PROGRAM OP90_MP_IO
VAR
	OP90_MP_DI_MODULE_1 AT %I* : WORD;
	OP90_MP_DI_MODULE_2 AT %I* : WORD;
	OP90_MP_DI_MODULE_3 AT %I* : WORD;
	
	OP90_MP_DO_MODULE_1 AT %Q* : WORD;
	OP90_MP_DO_MODULE_2 AT %Q* : WORD;
	
	WORD_AS_BIT_0: WORD_AS_BIT;
	WORD_AS_BIT_1: WORD_AS_BIT;
	WORD_AS_BIT_2: WORD_AS_BIT;
	
	BIT_AS_WORD_0: BIT_AS_WORD;
	BIT_AS_WORD_1: BIT_AS_WORD;
END_VAR

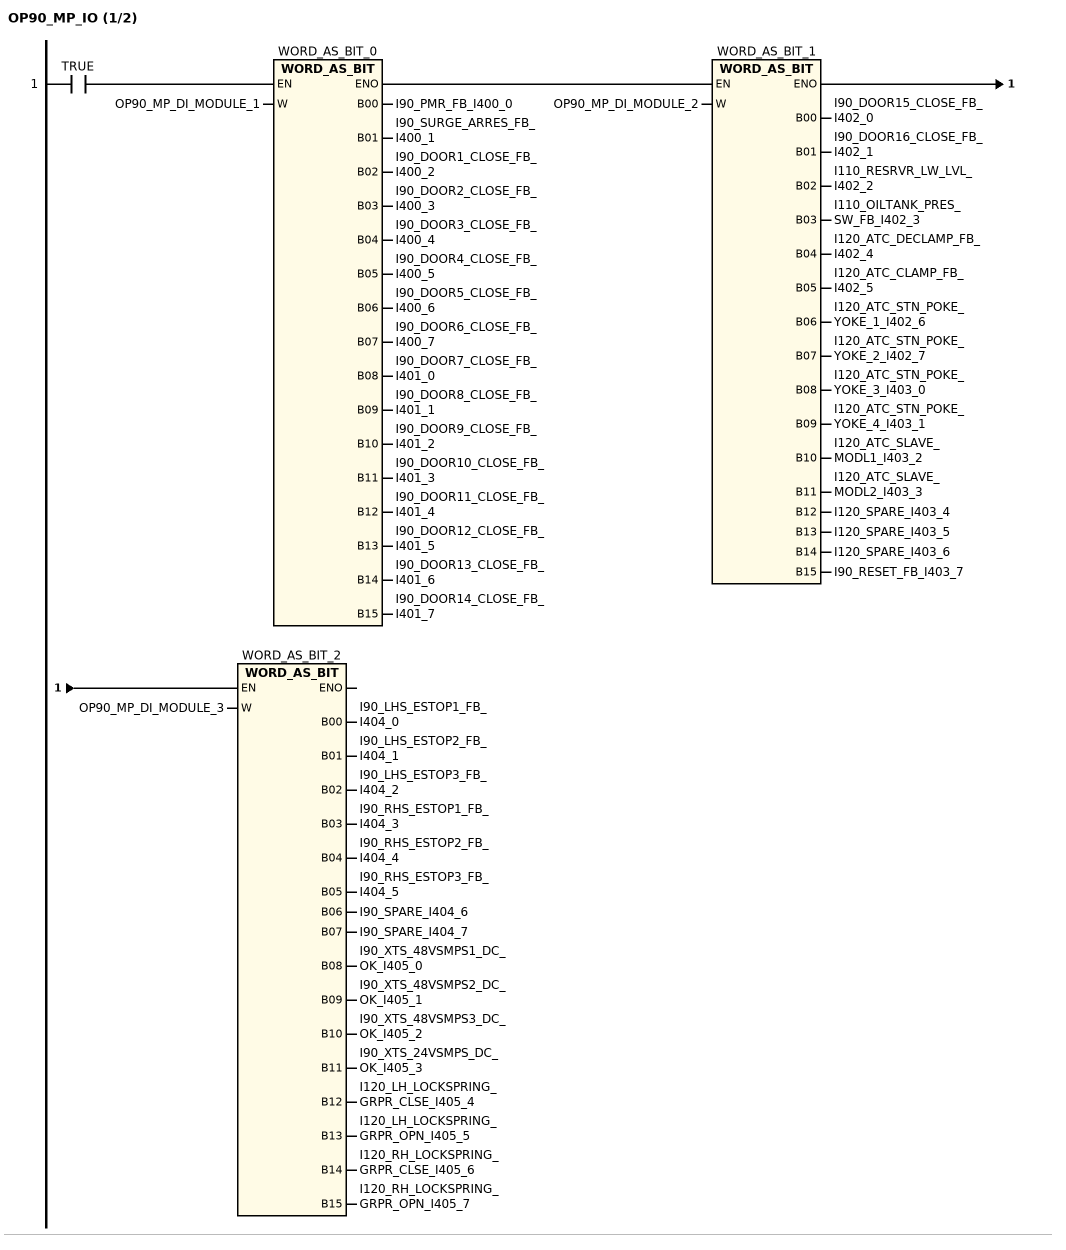
// NETWORK 1
WORD_AS_BIT_0(
    W := OP90_MP_DI_MODULE_1,
    B00 => I90_PMR_FB_I400_0,
    B01 => I90_SURGE_ARRES_FB_I400_1,
    B02 => I90_DOOR1_CLOSE_FB_I400_2,
    B03 => I90_DOOR2_CLOSE_FB_I400_3,
    B04 => I90_DOOR3_CLOSE_FB_I400_4,
    B05 => I90_DOOR4_CLOSE_FB_I400_5,
    B06 => I90_DOOR5_CLOSE_FB_I400_6,
    B07 => I90_DOOR6_CLOSE_FB_I400_7,
    B08 => I90_DOOR7_CLOSE_FB_I401_0,
    B09 => I90_DOOR8_CLOSE_FB_I401_1,
    B10 => I90_DOOR9_CLOSE_FB_I401_2,
    B11 => I90_DOOR10_CLOSE_FB_I401_3,
    B12 => I90_DOOR11_CLOSE_FB_I401_4,
    B13 => I90_DOOR12_CLOSE_FB_I401_5,
    B14 => I90_DOOR13_CLOSE_FB_I401_6,
    B15 => I90_DOOR14_CLOSE_FB_I401_7); // WORD_AS_BIT
WORD_AS_BIT_1(
    W := OP90_MP_DI_MODULE_2,
    B00 => I90_DOOR15_CLOSE_FB_I402_0,
    B01 => I90_DOOR16_CLOSE_FB_I402_1,
    B02 => I110_RESRVR_LW_LVL_I402_2,
    B03 => I110_OILTANK_PRES_SW_FB_I402_3,
    B04 => I120_ATC_DECLAMP_FB_I402_4,
    B05 => I120_ATC_CLAMP_FB_I402_5,
    B06 => I120_ATC_STN_POKE_YOKE_1_I402_6,
    B07 => I120_ATC_STN_POKE_YOKE_2_I402_7,
    B08 => I120_ATC_STN_POKE_YOKE_3_I403_0,
    B09 => I120_ATC_STN_POKE_YOKE_4_I403_1,
    B10 => I120_ATC_SLAVE_MODL1_I403_2,
    B11 => I120_ATC_SLAVE_MODL2_I403_3,
    B12 => I120_SPARE_I403_4,
    B13 => I120_SPARE_I403_5,
    B14 => I120_SPARE_I403_6,
    B15 => I90_RESET_FB_I403_7); // WORD_AS_BIT
WORD_AS_BIT_2(
    W := OP90_MP_DI_MODULE_3,
    B00 => I90_LHS_ESTOP1_FB_I404_0,
    B01 => I90_LHS_ESTOP2_FB_I404_1,
    B02 => I90_LHS_ESTOP3_FB_I404_2,
    B03 => I90_RHS_ESTOP1_FB_I404_3,
    B04 => I90_RHS_ESTOP2_FB_I404_4,
    B05 => I90_RHS_ESTOP3_FB_I404_5,
    B06 => I90_SPARE_I404_6,
    B07 => I90_SPARE_I404_7,
    B08 => I90_XTS_48VSMPS1_DC_OK_I405_0,
    B09 => I90_XTS_48VSMPS2_DC_OK_I405_1,
    B10 => I90_XTS_48VSMPS3_DC_OK_I405_2,
    B11 => I90_XTS_24VSMPS_DC_OK_I405_3,
    B12 => I120_LH_LOCKSPRING_GRPR_CLSE_I405_4,
    B13 => I120_LH_LOCKSPRING_GRPR_OPN_I405_5,
    B14 => I120_RH_LOCKSPRING_GRPR_CLSE_I405_6,
    B15 => I120_RH_LOCKSPRING_GRPR_OPN_I405_7); // WORD_AS_BIT

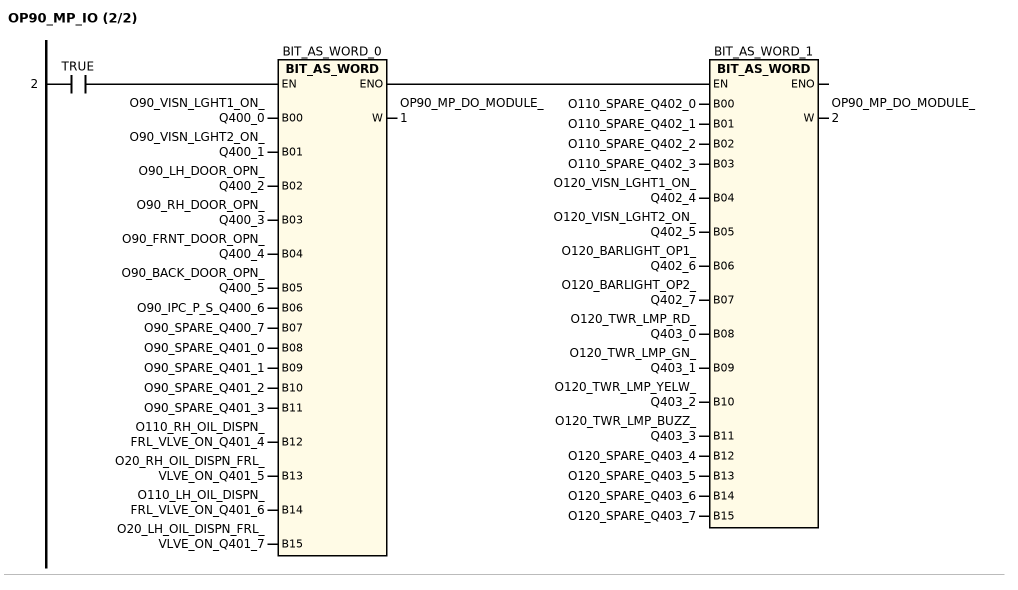
// NETWORK 2
BIT_AS_WORD_0(
    B00 := O90_VISN_LGHT1_ON_Q400_0,
    B01 := O90_VISN_LGHT2_ON_Q400_1,
    B02 := O90_LH_DOOR_OPN_Q400_2,
    B03 := O90_RH_DOOR_OPN_Q400_3,
    B04 := O90_FRNT_DOOR_OPN_Q400_4,
    B05 := O90_BACK_DOOR_OPN_Q400_5,
    B06 := O90_IPC_P_S_Q400_6,
    B07 := O90_SPARE_Q400_7,
    B08 := O90_SPARE_Q401_0,
    B09 := O90_SPARE_Q401_1,
    B10 := O90_SPARE_Q401_2,
    B11 := O90_SPARE_Q401_3,
    B12 := O110_RH_OIL_DISPN_FRL_VLVE_ON_Q401_4,
    B13 := O20_RH_OIL_DISPN_FRL_VLVE_ON_Q401_5,
    B14 := O110_LH_OIL_DISPN_FRL_VLVE_ON_Q401_6,
    B15 := O20_LH_OIL_DISPN_FRL_VLVE_ON_Q401_7,
    W => OP90_MP_DO_MODULE_1); // BIT_AS_WORD
BIT_AS_WORD_1(
    B00 := O110_SPARE_Q402_0,
    B01 := O110_SPARE_Q402_1,
    B02 := O110_SPARE_Q402_2,
    B03 := O110_SPARE_Q402_3,
    B04 := O120_VISN_LGHT1_ON_Q402_4,
    B05 := O120_VISN_LGHT2_ON_Q402_5,
    B06 := O120_BARLIGHT_OP1_Q402_6,
    B07 := O120_BARLIGHT_OP2_Q402_7,
    B08 := O120_TWR_LMP_RD_Q403_0,
    B09 := O120_TWR_LMP_GN_Q403_1,
    B10 := O120_TWR_LMP_YELW_Q403_2,
    B11 := O120_TWR_LMP_BUZZ_Q403_3,
    B12 := O120_SPARE_Q403_4,
    B13 := O120_SPARE_Q403_5,
    B14 := O120_SPARE_Q403_6,
    B15 := O120_SPARE_Q403_7,
    W => OP90_MP_DO_MODULE_2); // BIT_AS_WORD

END_PROGRAM

(* stored: Version 1.1.0.1, ProductVersion 3.1.4024.11
   POU OP90_MP_IO: Id {5d8eaf86-6a03-4884-a501-213b6b4be573}, SpecialFunc None *)
